# EPICS substitutions: superlogicsSup/superlogics_thermo_connected.substitutions
file superlogics_thermo_connected.template {
    pattern {CHNL}

    {"0"}
    {"1"}
    {"2"}
    {"3"}
    {"4"}
    {"5"}
    {"6"}
    {"7"}
}
